   A_22_A800Z1.CmdRstTrueTime := FALSE;
   A_22_A800Z1.CmdRstFalseTime := FALSE;
   A_22_A800Z1.CmdRunTimeoutTime := FALSE;
   A_22_A800Z1.CmdFaultReset := FALSE;
   A_22_A800Z1.InLocal := FALSE;
   A_22_A800Z1.spare0305 := FALSE;
   A_22_A800Z1.InReport := FALSE;
   A_22_A800Z1.OutTimeoutTime := FALSE;
   A_22_A800Z1.InHWStop := FALSE;
   A_22_A800Z1.InDPFault := FALSE;
   A_22_A800Z1.OutPreAlarmTrue := FALSE;
   A_22_A800Z1.OutPreAlarmFalse := FALSE;
   A_22_A800Z1.OutFlagPos := FALSE;
   A_22_A800Z1.OutFlagNeg := FALSE;
   A_22_A800Z1.OutpFaultReset := FALSE;
   A_22_A800Z1.OutTrue := FALSE;
   A_22_A800Z1.StFalse := FALSE;
   A_22_A800Z1.StCtoTrue := FALSE;
   A_22_A800Z1.StTrue := FALSE;
   A_22_A800Z1.StCtoFalse := FALSE;
   A_22_A800Z1.StFault := FALSE;
   A_22_A800Z1.OutAlarmNrLog := 0;
   A_22_A800Z1.Par.ParObjectNo := 0;
   A_22_A800Z1.Par.ParMsgType := 0;
   A_22_A800Z1.Par.ParHornCode := 0;
   A_22_A800Z1.Par.ParLogOff := FALSE;
   A_22_A800Z1.Par.spare0401 := FALSE;
   A_22_A800Z1.Par.Par2WorkingCond := FALSE;
   A_22_A800Z1.Par.ParFaultRetry := FALSE;
   A_22_A800Z1.Par.ParBinLevel := FALSE;
   A_22_A800Z1.Par.ParDelayChange := 0;
   A_22_A800Z1.Par.ParDelayTrue := 0;
   A_22_A800Z1.Par.ParDelayFalse := 0;
   A_22_A800Z1.Par.ParTimeoutTrue := 0;
   A_22_A800Z1.Par.ParTimeoutFalse := 0;
   A_22_A800Z1.Par.OutMonTime := 0;
   A_22_A800Z1.Par.OutTransitionTime := 0;
   A_22_A800Z1.Par.OutMonTrue := FALSE;
   A_22_A800Z1.Par.OutMonFalse := FALSE;
   A_22_A800Z1.Par.OutFlagFaultDev := FALSE;
   A_22_A800Z1.Par.OutDelayTime := 0;
//Parameter =A-22-A106Z1 : EMERGENCY STOP FROM +C21
      #A_22_A106Z1.Par.ParObjectNo                             :=635;
      #A_22_A106Z1.Par.ParMsgType                              :=7171;
      #A_22_A106Z1.Par.ParHornCode                             :=2;
      #A_22_A106Z1.Par.ParDelayChange                          :=0;
      #A_22_A106Z1.Par.ParDelayTrue                            :=10;
      #A_22_A106Z1.Par.ParDelayFalse                           :=0;
      #A_22_A106Z1.Par.ParTimeoutTrue                          :=0;
      #A_22_A106Z1.Par.ParTimeoutFalse                         :=0;
      #A_22_A106Z1.Par.ParLogOff                               :=False;
      #A_22_A106Z1.Par.Par2WorkingCond                         :=False;
      #A_22_A106Z1.Par.ParFaultRetry                           :=False;
      #A_22_A106Z1.Par.ParBinLevel                             :=False;
//
//
END_DATA_BLOCK

